INTERFACE I_ForcibleBool EXTENDS I_Base

{attribute 'monitoring' := 'call'}
PROPERTY Force : E_ForceState
GET
END_GET
SET
END_SET
END_PROPERTY

END_INTERFACE

(* stored: Version 1.1.0.1, ProductVersion 3.1.4026.18
   Itf I_ForcibleBool: Id {56bd5c6a-00f8-4316-ab2a-af3720b8bb94}
   Property Force: Id {4b636602-23e9-42ab-a6d6-0ad9c07ec265}
   Get Get: Id {b2b6ea85-c67a-416b-9746-3a00644a4436}
   Set Set: Id {5de82df9-eaf5-44b2-b95d-1a9a1eb1dc20} *)
